Yaskawa INFORM job: TESTR22.JBI

/JOB
//NAME TESTR22
///FOLDERNAME INNE
//POS
///NPOS 12,12,12,0,0,0
///TOOL 0
///POSTYPE PULSE
///PULSE
C00000=26806,-11126,4152,28099,80822,-32630
C00001=26783,-11151,4133,28099,80829,-32637
C00002=26780,-11154,4131,28099,80829,-32638
C00003=26779,-11156,4130,28099,80830,-32638
C00004=26719,-11509,2564,28050,81544,-32488
C00005=26170,-11851,2534,28047,81587,-32686
C00006=26786,-11150,4134,28098,80828,-32636
C00007=26999,-10988,4259,28103,80762,-32571
C00008=27006,-10982,4263,28103,80760,-32569
C00009=27007,-10981,4264,28103,80760,-32568
C00010=27009,-10978,4267,28104,80759,-32567
C00011=27033,-10953,4286,28104,80752,-32560
BC00000=274902,1351538,800161
BC00001=274902,1351538,692627
BC00002=273972,1345884,674703
BC00003=273600,1343622,667533
BC00004=273600,1343622,667533
BC00005=273600,1343622,667533
BC00006=268892,1343625,670294
BC00007=121534,1343738,756653
BC00008=116826,1343743,759410
BC00009=117198,1346004,766579
BC00010=118128,1351658,784503
BC00011=118128,1351658,892038
EC00000=0,0
EC00001=0,0
EC00002=0,0
EC00003=0,0
EC00004=0,0
EC00005=0,0
EC00006=0,0
EC00007=0,0
EC00008=0,0
EC00009=0,0
EC00010=0,0
EC00011=0,0
//INST
///DATE 2023/10/04 15:12
///ATTR SC,RW
///GROUP1 RB1,BS1
///GROUP2 ST1
NOP
'TESTr22
'Path W701
SSFTOF
MOVJ C00000 BC00000 VJ=100.00  +MOVJ EC00000 VJ=100.00
MOVL C00001 BC00001 V=1000.0  +MOVJ EC00001 VJ=100.00
MOVL C00002 BC00002 V=400.0  +MOVJ EC00002 VJ=100.00
SMOVL C00003 BC00003 V=100.0 PL=0  +MOVJ EC00003
SREFP 1 C00004 BC00004  +REFP EC00004
SREFP 2 C00005 BC00005  +REFP EC00005
SMOVL C00006 BC00006 V=10.0  +MOVJ EC00006
SMOVL C00007 BC00007 V=10.0  +MOVJ EC00007
SMOVL C00008 BC00008 V=10.0  +MOVJ EC00008
MOVL C00009 BC00009 V=400.0  +MOVJ EC00009 VJ=100.00
MOVL C00010 BC00010 V=1000.0  +MOVJ EC00010 VJ=100.00
MOVL C00011 BC00011 V=1000.0  +MOVJ EC00011 VJ=100.00
END
